// TIA Portal V16 export
// export: Created 2022-11-17T15:49:33.7252465Z, ExportSetting WithDefaults, DisplayName Totally Integrated Automation Portal, DisplayVersion V16 Update 6, DisplayName TIA Portal Version Control Interface, DisplayVersion V16 Update 2, DisplayName TIA Portal Openness, DisplayVersion V16 Update 6, DisplayName SINAMICS Startdrive Advanced, DisplayVersion V16 Update 5, DisplayName SINAMICS Startdrive G130, G150, S120, S150, SINAMICS MV, S210, DisplayVersion V16 Update 5, DisplayName SINAMICS Startdrive G110M, G120, G120C, G120D, G120P, G115D, DisplayVersion V16 Update 5, DisplayName STEP 7 Professional, DisplayVersion V16 Update 6, DisplayName STEP 7 Safety, DisplayVersion V16, DisplayName WinCC Advanced, DisplayVersion V16 Update 6
ORGANIZATION_BLOCK "Main"   // OB1, LAD, ProgramCycle
TITLE = "Main Program Sweep (Cycle)"
{ S7_Optimized_Access := 'TRUE' }
VERSION : 0.1
// stored: AutoNumber false, IsIECCheckEnabled false, SetENOAutomatically false
   VAR_TEMP
      SALDATORE : Bool;
      PORTA : Bool;
      ESAUR_FILM : Bool;
      STR_FASCIA : Bool;
      STR_CORDA : Bool;
      CONTRASTO : Bool;
      PRESSORE : Bool;
      PRESS_RECT : Bool;
      AUTO_CENTR : Bool;
      TOP : Bool;
      BRAKE : Bool;   // Table phase
      PHASE : Bool;   // Table brake
   END_VAR
   VAR_TEMP   // added for the SCL form of the ladder/FBD networks
      _w1 : Bool;
      _w2 : Bool;
      _w3 : Bool;
   END_VAR
BEGIN

REGION Network 1: Bit always on
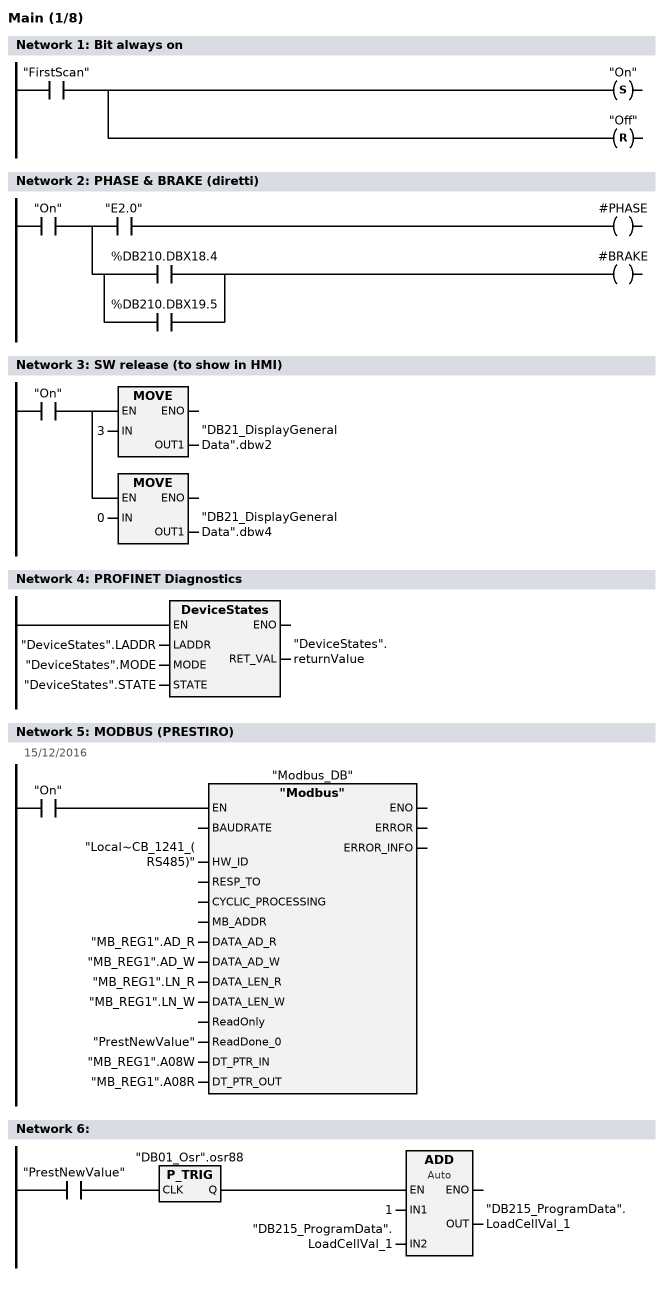
   RUNG wire#powerrail
      Contact( "FirstScan" )
      wire#w1
      S_Coil( "On" )
   END_RUNG
   RUNG wire#w1
      R_Coil( "Off" )
   END_RUNG
   // the same network as SCL:
   IF "FirstScan" THEN
       "On" := TRUE;
       "Off" := FALSE;
   END_IF;
END_REGION

REGION Network 2: PHASE & BRAKE (diretti)
   RUNG wire#powerrail
      Contact( "On" )
      wire#w1
      Contact( "E2.0" )
      Coil( #PHASE )
   END_RUNG
   RUNG wire#w1
      Contact( %DB210.DBX18.4 )
      wire#w2
      Coil( #BRAKE )
   END_RUNG
   RUNG wire#w1
      Contact( %DB210.DBX19.5 )
   END_RUNG wire#w2
   // the same network as SCL:
   #PHASE := "On" AND "E2.0";
   #BRAKE := "On" AND (%DB210.DBX18.4 OR %DB210.DBX19.5);
END_REGION

REGION Network 3: SW release (to show in HMI)
   RUNG wire#powerrail
      Contact( "On" )
      wire#w1
      Move(in := 3, out1 => "DB21_DisplayGeneralData".dbw2)
   END_RUNG
   RUNG wire#w1
      Move(in := 0, out1 => "DB21_DisplayGeneralData".dbw4)
   END_RUNG
   // the same network as SCL:
   IF "On" THEN
       "DB21_DisplayGeneralData".dbw2 := 3;
       "DB21_DisplayGeneralData".dbw4 := 0;
   END_IF;
END_REGION

REGION Network 4: PROFINET Diagnostics
   RUNG wire#powerrail
      DeviceStates(LADDR := "DeviceStates".LADDR, MODE := "DeviceStates".MODE, STATE := "DeviceStates".STATE, Ret_Val => "DeviceStates".returnValue)
   END_RUNG
   // the same network as SCL:
   "DeviceStates".returnValue := DeviceStates(LADDR := "DeviceStates".LADDR,
                           MODE := "DeviceStates".MODE,
                           STATE := "DeviceStates".STATE);
END_REGION

REGION Network 5: MODBUS (PRESTIRO)
   // 15/12/2016
   RUNG wire#powerrail
      Contact( "On" )
      "Modbus_DB"(BAUDRATE :=, HW_ID := "Local~CB_1241_(RS485)", RESP_TO :=, CYCLIC_PROCESSING :=, MB_ADDR :=, DATA_AD_R := "MB_REG1".AD_R, DATA_AD_W := "MB_REG1".AD_W, DATA_LEN_R := "MB_REG1".LN_R, DATA_LEN_W := "MB_REG1".LN_W, ReadOnly :=, ReadDone_0 := "PrestNewValue", DT_PTR_IN := "MB_REG1".A08W, DT_PTR_OUT := "MB_REG1".A08R, ERROR =>, ERROR_INFO =>)
   END_RUNG
   // the same network as SCL:
   IF "On" THEN
       "Modbus_DB"(HW_ID := "Local~CB_1241_(RS485)",   // "Modbus"
                   DATA_AD_R := "MB_REG1".AD_R,
                   DATA_AD_W := "MB_REG1".AD_W,
                   DATA_LEN_R := "MB_REG1".LN_R,
                   DATA_LEN_W := "MB_REG1".LN_W,
                   ReadDone_0 := "PrestNewValue",
                   DT_PTR_IN := "MB_REG1".A08W,
                   DT_PTR_OUT := "MB_REG1".A08R);
   END_IF;
END_REGION

REGION Network 6
   RUNG wire#powerrail
      Contact( "PrestNewValue" )
      P_Trig( "DB01_Osr".osr88 )
      Add(in1 := 1, in2 := "DB215_ProgramData".LoadCellVal_1, out => "DB215_ProgramData".LoadCellVal_1)
   END_RUNG
   // the same network as SCL:
   #_w1 := "PrestNewValue" AND NOT "DB01_Osr".osr88;   // rising edge
   "DB01_Osr".osr88 := "PrestNewValue";
   IF #_w1 THEN "DB215_ProgramData".LoadCellVal_1 := 1 + "DB215_ProgramData".LoadCellVal_1; END_IF;
END_REGION

REGION Network 7: Reset Modbus errors
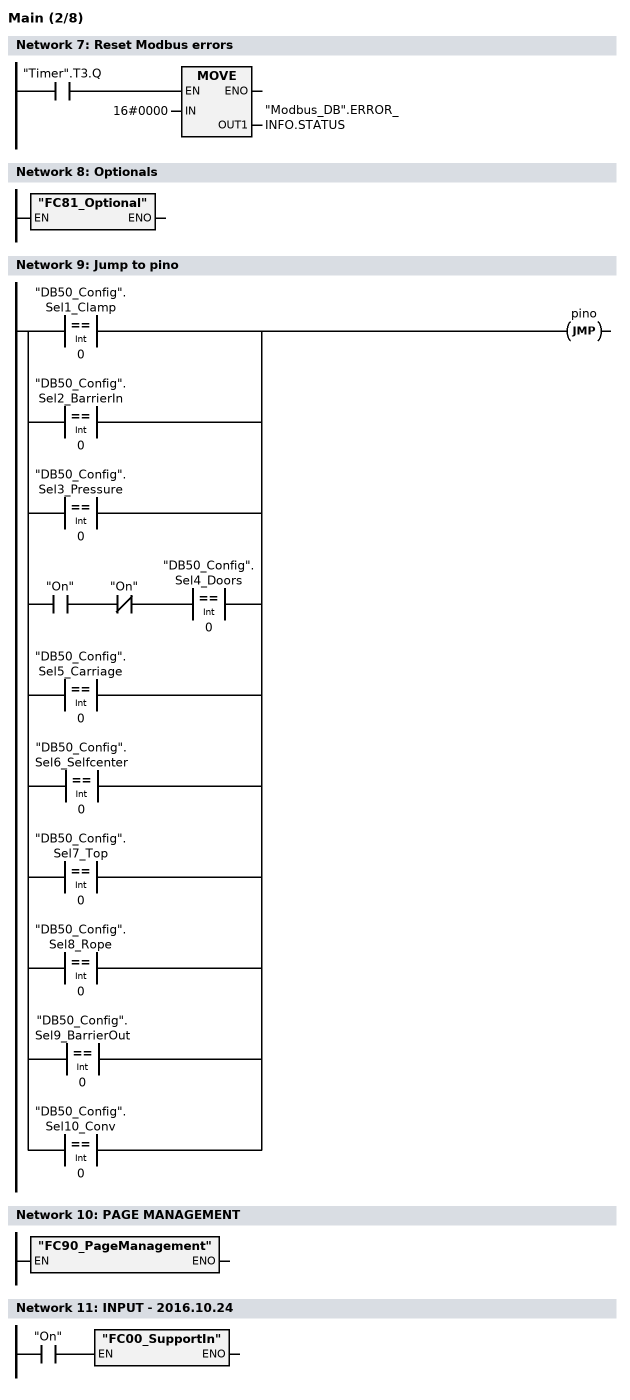
   RUNG wire#powerrail
      Contact( "Timer".T3.Q )
      Move(in := 16#0000, out1 => "Modbus_DB".ERROR_INFO.STATUS)
   END_RUNG
   // the same network as SCL:
   IF "Timer".T3.Q THEN "Modbus_DB".ERROR_INFO.STATUS := 16#0000; END_IF;
END_REGION

REGION Network 8: Optionals
   RUNG wire#powerrail
      "FC81_Optional"()
   END_RUNG
   // the same network as SCL:
   "FC81_Optional"();
END_REGION

REGION Network 9: Jump to pino
   RUNG wire#powerrail
      { S7_Templates := "SrcType := Int" } EQ_Contact(in1 := "DB50_Config".Sel1_Clamp, in2 := 0)
      wire#w1
      JumpCoil( pino )
   END_RUNG
   RUNG wire#powerrail
      { S7_Templates := "SrcType := Int" } EQ_Contact(in1 := "DB50_Config".Sel2_BarrierIn, in2 := 0)
   END_RUNG wire#w1
   RUNG wire#powerrail
      { S7_Templates := "SrcType := Int" } EQ_Contact(in1 := "DB50_Config".Sel3_Pressure, in2 := 0)
   END_RUNG wire#w1
   RUNG wire#powerrail
      Contact( "On" )
      I_Contact( "On" )
      { S7_Templates := "SrcType := Int" } EQ_Contact(in1 := "DB50_Config".Sel4_Doors, in2 := 0)
   END_RUNG wire#w1
   RUNG wire#powerrail
      { S7_Templates := "SrcType := Int" } EQ_Contact(in1 := "DB50_Config".Sel5_Carriage, in2 := 0)
   END_RUNG wire#w1
   RUNG wire#powerrail
      { S7_Templates := "SrcType := Int" } EQ_Contact(in1 := "DB50_Config".Sel6_Selfcenter, in2 := 0)
   END_RUNG wire#w1
   RUNG wire#powerrail
      { S7_Templates := "SrcType := Int" } EQ_Contact(in1 := "DB50_Config".Sel7_Top, in2 := 0)
   END_RUNG wire#w1
   RUNG wire#powerrail
      { S7_Templates := "SrcType := Int" } EQ_Contact(in1 := "DB50_Config".Sel8_Rope, in2 := 0)
   END_RUNG wire#w1
   RUNG wire#powerrail
      { S7_Templates := "SrcType := Int" } EQ_Contact(in1 := "DB50_Config".Sel9_BarrierOut, in2 := 0)
   END_RUNG wire#w1
   RUNG wire#powerrail
      { S7_Templates := "SrcType := Int" } EQ_Contact(in1 := "DB50_Config".Sel10_Conv, in2 := 0)
   END_RUNG wire#w1
   // the same network as SCL:
   IF ("DB50_Config".Sel1_Clamp = 0) OR ("DB50_Config".Sel2_BarrierIn = 0) OR ("DB50_Config".Sel3_Pressure = 0) OR ("On" AND NOT "On" AND ("DB50_Config".Sel4_Doors = 0)) OR ("DB50_Config".Sel5_Carriage = 0) OR ("DB50_Config".Sel6_Selfcenter = 0) OR ("DB50_Config".Sel7_Top = 0) OR ("DB50_Config".Sel8_Rope = 0) OR ("DB50_Config".Sel9_BarrierOut = 0) OR ("DB50_Config".Sel10_Conv = 0) THEN
       GOTO pino;
   END_IF;
END_REGION

REGION Network 10: PAGE MANAGEMENT
   RUNG wire#powerrail
      "FC90_PageManagement"()
   END_RUNG
   // the same network as SCL:
   "FC90_PageManagement"();
END_REGION

REGION Network 11: INPUT - 2016.10.24
   RUNG wire#powerrail
      Contact( "On" )
      "FC00_SupportIn"()
   END_RUNG
   // the same network as SCL:
   IF "On" THEN "FC00_SupportIn"(); END_IF;
END_REGION

REGION Network 12: ACCESSORIES (CONFIGURATION)
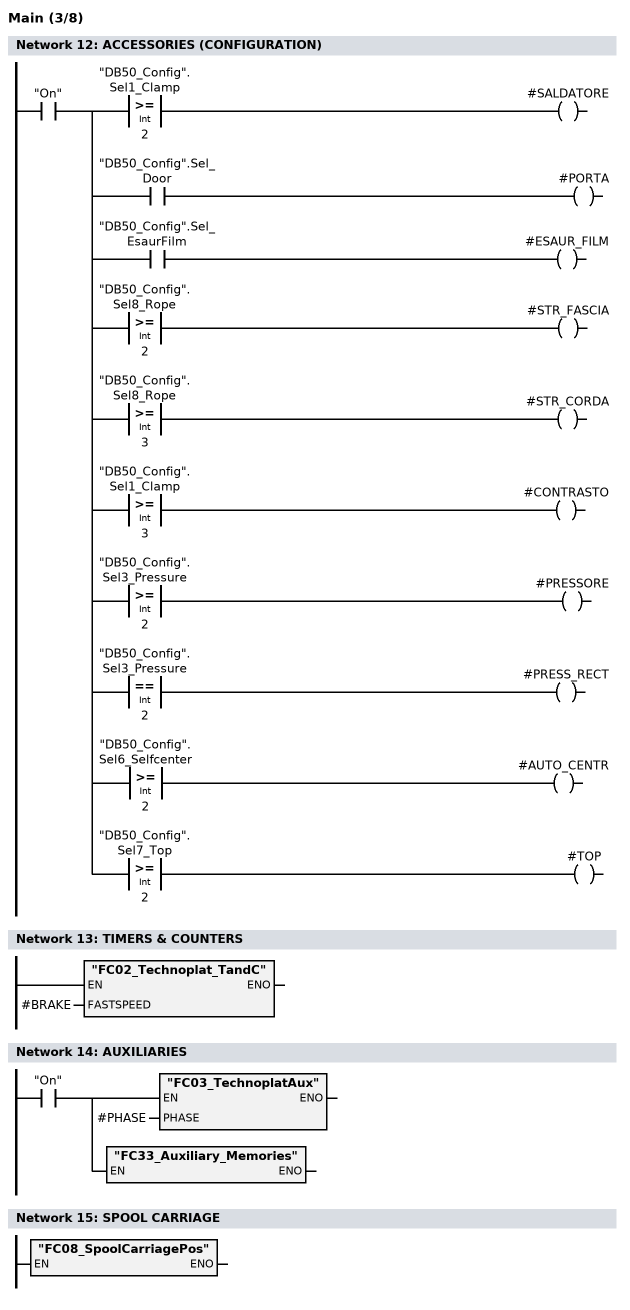
   RUNG wire#powerrail
      Contact( "On" )
      wire#w1
      { S7_Templates := "SrcType := Int" } GE_Contact(in1 := "DB50_Config".Sel1_Clamp, in2 := 2)
      Coil( #SALDATORE )
   END_RUNG
   RUNG wire#w1
      Contact( "DB50_Config".Sel_Door )
      Coil( #PORTA )
   END_RUNG
   RUNG wire#w1
      Contact( "DB50_Config".Sel_EsaurFilm )
      Coil( #ESAUR_FILM )
   END_RUNG
   RUNG wire#w1
      { S7_Templates := "SrcType := Int" } GE_Contact(in1 := "DB50_Config".Sel8_Rope, in2 := 2)
      Coil( #STR_FASCIA )
   END_RUNG
   RUNG wire#w1
      { S7_Templates := "SrcType := Int" } GE_Contact(in1 := "DB50_Config".Sel8_Rope, in2 := 3)
      Coil( #STR_CORDA )
   END_RUNG
   RUNG wire#w1
      { S7_Templates := "SrcType := Int" } GE_Contact(in1 := "DB50_Config".Sel1_Clamp, in2 := 3)
      Coil( #CONTRASTO )
   END_RUNG
   RUNG wire#w1
      { S7_Templates := "SrcType := Int" } GE_Contact(in1 := "DB50_Config".Sel3_Pressure, in2 := 2)
      Coil( #PRESSORE )
   END_RUNG
   RUNG wire#w1
      { S7_Templates := "SrcType := Int" } EQ_Contact(in1 := "DB50_Config".Sel3_Pressure, in2 := 2)
      Coil( #PRESS_RECT )
   END_RUNG
   RUNG wire#w1
      { S7_Templates := "SrcType := Int" } GE_Contact(in1 := "DB50_Config".Sel6_Selfcenter, in2 := 2)
      Coil( #AUTO_CENTR )
   END_RUNG
   RUNG wire#w1
      { S7_Templates := "SrcType := Int" } GE_Contact(in1 := "DB50_Config".Sel7_Top, in2 := 2)
      Coil( #TOP )
   END_RUNG
   // the same network as SCL:
   #SALDATORE := "On" AND ("DB50_Config".Sel1_Clamp >= 2);
   #PORTA := "On" AND "DB50_Config".Sel_Door;
   #ESAUR_FILM := "On" AND "DB50_Config".Sel_EsaurFilm;
   #STR_FASCIA := "On" AND ("DB50_Config".Sel8_Rope >= 2);
   #STR_CORDA := "On" AND ("DB50_Config".Sel8_Rope >= 3);
   #CONTRASTO := "On" AND ("DB50_Config".Sel1_Clamp >= 3);
   #PRESSORE := "On" AND ("DB50_Config".Sel3_Pressure >= 2);
   #PRESS_RECT := "On" AND ("DB50_Config".Sel3_Pressure = 2);
   #AUTO_CENTR := "On" AND ("DB50_Config".Sel6_Selfcenter >= 2);
   #TOP := "On" AND ("DB50_Config".Sel7_Top >= 2);
END_REGION

REGION Network 13: TIMERS & COUNTERS
   RUNG wire#powerrail
      "FC02_Technoplat_TandC"(FASTSPEED := #BRAKE)
   END_RUNG
   // the same network as SCL:
   "FC02_Technoplat_TandC"(FASTSPEED := #BRAKE);
END_REGION

REGION Network 14: AUXILIARIES
   RUNG wire#powerrail
      Contact( "On" )
      wire#w1
      "FC03_TechnoplatAux"(PHASE := #PHASE)
   END_RUNG
   RUNG wire#w1
      "FC33_Auxiliary_Memories"()
   END_RUNG
   // the same network as SCL:
   #_w1 := "On";
   IF #_w1 THEN
       "FC03_TechnoplatAux"(PHASE := #PHASE);
       "FC33_Auxiliary_Memories"();
   END_IF;
END_REGION

REGION Network 15: SPOOL CARRIAGE
   RUNG wire#powerrail
      "FC08_SpoolCarriagePos"()
   END_RUNG
   // the same network as SCL:
   "FC08_SpoolCarriagePos"();
END_REGION

REGION Network 16: ROTATION TABLE
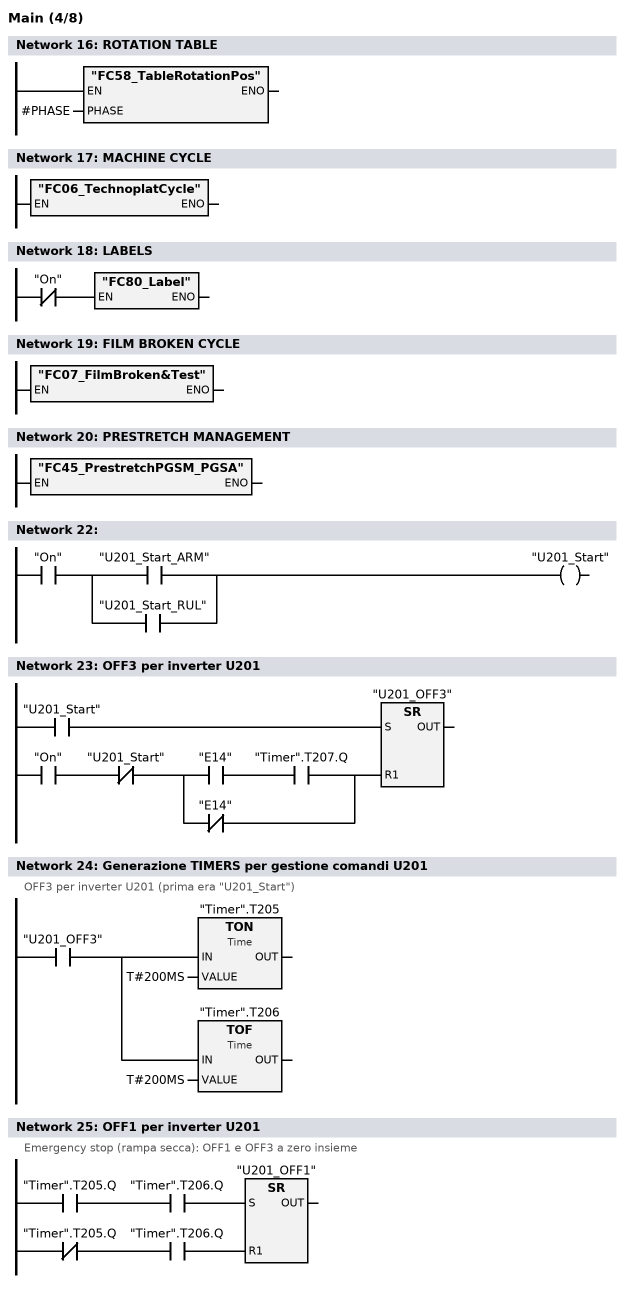
   RUNG wire#powerrail
      "FC58_TableRotationPos"(PHASE := #PHASE)
   END_RUNG
   // the same network as SCL:
   "FC58_TableRotationPos"(PHASE := #PHASE);
END_REGION

REGION Network 17: MACHINE CYCLE
   RUNG wire#powerrail
      "FC06_TechnoplatCycle"()
   END_RUNG
   // the same network as SCL:
   "FC06_TechnoplatCycle"();
END_REGION

REGION Network 18: LABELS
   RUNG wire#powerrail
      I_Contact( "On" )
      "FC80_Label"()
   END_RUNG
   // the same network as SCL:
   IF NOT "On" THEN "FC80_Label"(); END_IF;
END_REGION

REGION Network 19: FILM BROKEN CYCLE
   RUNG wire#powerrail
      "FC07_FilmBroken&Test"()
   END_RUNG
   // the same network as SCL:
   "FC07_FilmBroken&Test"();
END_REGION

REGION Network 20: PRESTRETCH MANAGEMENT
   RUNG wire#powerrail
      "FC45_PrestretchPGSM_PGSA"()
   END_RUNG
   // the same network as SCL:
   "FC45_PrestretchPGSM_PGSA"();
END_REGION

REGION Network 21: - - - GESTIONE INVERTER PROFINET - - -
END_REGION

REGION Network 22
   RUNG wire#powerrail
      Contact( "On" )
      wire#w1
      Contact( "U201_Start_ARM" )
      wire#w2
      Coil( "U201_Start" )
   END_RUNG
   RUNG wire#w1
      Contact( "U201_Start_RUL" )
   END_RUNG wire#w2
   // the same network as SCL:
   "U201_Start" := "On" AND ("U201_Start_ARM" OR "U201_Start_RUL");
END_REGION

REGION Network 23: OFF3 per inverter U201
   RUNG wire#powerrail
      Contact( "U201_Start" )
      S_SR(operand := "U201_OFF3", r1 := wire#w2)
   END_RUNG
   RUNG wire#powerrail
      Contact( "On" )
      I_Contact( "U201_Start" )
      wire#w1
      Contact( "E14" )
      Contact( "Timer".T207.Q )
   END_RUNG wire#w2
   RUNG wire#w1
      I_Contact( "E14" )
   END_RUNG wire#w2
   // the same network as SCL:
   IF "U201_Start" THEN
       "U201_OFF3" := TRUE;   // SR flip-flop
   END_IF;
   IF "On" AND NOT "U201_Start" AND (("E14" AND "Timer".T207.Q) OR NOT "E14") THEN
       "U201_OFF3" := FALSE;
   END_IF;
END_REGION

REGION Network 24: Generazione TIMERS per gestione comandi U201
   // OFF3 per inverter U201 (prima era "U201_Start")
   "Timer".T205.TON(IN := "U201_OFF3", PT := T#200MS);   // TON coil
   "Timer".T206.TOF(IN := "U201_OFF3", PT := T#200MS);   // TOF coil
END_REGION

REGION Network 25: OFF1 per inverter U201
   // Emergency stop (rampa secca): OFF1 e OFF3 a zero insieme
   RUNG wire#powerrail
      Contact( "Timer".T205.Q )
      Contact( "Timer".T206.Q )
      S_SR(operand := "U201_OFF1", r1 := wire#w1)
   END_RUNG
   RUNG wire#powerrail
      I_Contact( "Timer".T205.Q )
      Contact( "Timer".T206.Q )
   END_RUNG wire#w1
   // the same network as SCL:
   IF "Timer".T205.Q AND "Timer".T206.Q THEN
       "U201_OFF1" := TRUE;   // SR flip-flop
   END_IF;
   IF NOT "Timer".T205.Q AND "Timer".T206.Q THEN "U201_OFF1" := FALSE; END_IF;
END_REGION

REGION Network 26: U201 - ROTAZIONE + CM
   // "U201_OFF1"/"U201_OFF3"
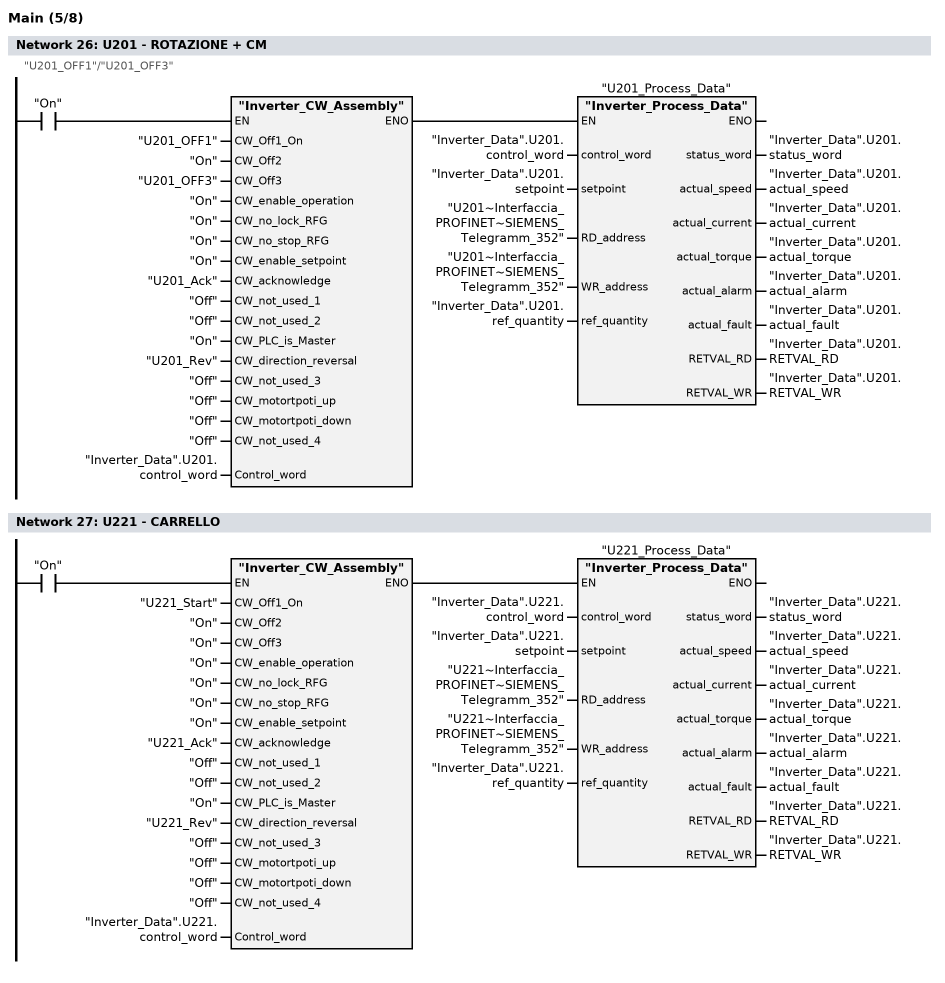
   RUNG wire#powerrail
      Contact( "On" )
      "Inverter_CW_Assembly"(CW_Off1_On := "U201_OFF1", CW_Off2 := "On", CW_Off3 := "U201_OFF3", CW_enable_operation := "On", CW_no_lock_RFG := "On", CW_no_stop_RFG := "On", CW_enable_setpoint := "On", CW_acknowledge := "U201_Ack", CW_not_used_1 := "Off", CW_not_used_2 := "Off", CW_PLC_is_Master := "On", CW_direction_reversal := "U201_Rev", CW_not_used_3 := "Off", CW_motortpoti_up := "Off", CW_motortpoti_down := "Off", CW_not_used_4 := "Off", Control_word := "Inverter_Data".U201.control_word)
      "U201_Process_Data"(control_word := "Inverter_Data".U201.control_word, setpoint := "Inverter_Data".U201.setpoint, RD_address := "U201~Interfaccia_PROFINET~SIEMENS_Telegramm_352", WR_address := "U201~Interfaccia_PROFINET~SIEMENS_Telegramm_352", ref_quantity := "Inverter_Data".U201.ref_quantity, status_word => "Inverter_Data".U201.status_word, actual_speed => "Inverter_Data".U201.actual_speed, actual_current => "Inverter_Data".U201.actual_current, actual_torque => "Inverter_Data".U201.actual_torque, actual_alarm => "Inverter_Data".U201.actual_alarm, actual_fault => "Inverter_Data".U201.actual_fault, RETVAL_RD => "Inverter_Data".U201.RETVAL_RD, RETVAL_WR => "Inverter_Data".U201.RETVAL_WR)
   END_RUNG
   // the same network as SCL:
   "Inverter_CW_Assembly"(EN := "On",
                          CW_Off1_On := "U201_OFF1",
                          CW_Off2 := "On",
                          CW_Off3 := "U201_OFF3",
                          CW_enable_operation := "On",
                          CW_no_lock_RFG := "On",
                          CW_no_stop_RFG := "On",
                          CW_enable_setpoint := "On",
                          CW_acknowledge := "U201_Ack",
                          CW_not_used_1 := "Off",
                          CW_not_used_2 := "Off",
                          CW_PLC_is_Master := "On",
                          CW_direction_reversal := "U201_Rev",
                          CW_not_used_3 := "Off",
                          CW_motortpoti_up := "Off",
                          CW_motortpoti_down := "Off",
                          CW_not_used_4 := "Off",
                          Control_word := "Inverter_Data".U201.control_word,
                          ENO => #_w1);
   IF #_w1 THEN
       "U201_Process_Data"(control_word := "Inverter_Data".U201.control_word,   // "Inverter_Process_Data"
                           setpoint := "Inverter_Data".U201.setpoint,
                           RD_address := "U201~Interfaccia_PROFINET~SIEMENS_Telegramm_352",
                           WR_address := "U201~Interfaccia_PROFINET~SIEMENS_Telegramm_352",
                           ref_quantity := "Inverter_Data".U201.ref_quantity,
                           status_word => "Inverter_Data".U201.status_word,
                           actual_speed => "Inverter_Data".U201.actual_speed,
                           actual_current => "Inverter_Data".U201.actual_current,
                           actual_torque => "Inverter_Data".U201.actual_torque,
                           actual_alarm => "Inverter_Data".U201.actual_alarm,
                           actual_fault => "Inverter_Data".U201.actual_fault,
                           RETVAL_RD => "Inverter_Data".U201.RETVAL_RD,
                           RETVAL_WR => "Inverter_Data".U201.RETVAL_WR);
   END_IF;
END_REGION

REGION Network 27: U221 - CARRELLO
   RUNG wire#powerrail
      Contact( "On" )
      "Inverter_CW_Assembly"(CW_Off1_On := "U221_Start", CW_Off2 := "On", CW_Off3 := "On", CW_enable_operation := "On", CW_no_lock_RFG := "On", CW_no_stop_RFG := "On", CW_enable_setpoint := "On", CW_acknowledge := "U221_Ack", CW_not_used_1 := "Off", CW_not_used_2 := "Off", CW_PLC_is_Master := "On", CW_direction_reversal := "U221_Rev", CW_not_used_3 := "Off", CW_motortpoti_up := "Off", CW_motortpoti_down := "Off", CW_not_used_4 := "Off", Control_word := "Inverter_Data".U221.control_word)
      "U221_Process_Data"(control_word := "Inverter_Data".U221.control_word, setpoint := "Inverter_Data".U221.setpoint, RD_address := "U221~Interfaccia_PROFINET~SIEMENS_Telegramm_352", WR_address := "U221~Interfaccia_PROFINET~SIEMENS_Telegramm_352", ref_quantity := "Inverter_Data".U221.ref_quantity, status_word => "Inverter_Data".U221.status_word, actual_speed => "Inverter_Data".U221.actual_speed, actual_current => "Inverter_Data".U221.actual_current, actual_torque => "Inverter_Data".U221.actual_torque, actual_alarm => "Inverter_Data".U221.actual_alarm, actual_fault => "Inverter_Data".U221.actual_fault, RETVAL_RD => "Inverter_Data".U221.RETVAL_RD, RETVAL_WR => "Inverter_Data".U221.RETVAL_WR)
   END_RUNG
   // the same network as SCL:
   "Inverter_CW_Assembly"(EN := "On",
                          CW_Off1_On := "U221_Start",
                          CW_Off2 := "On",
                          CW_Off3 := "On",
                          CW_enable_operation := "On",
                          CW_no_lock_RFG := "On",
                          CW_no_stop_RFG := "On",
                          CW_enable_setpoint := "On",
                          CW_acknowledge := "U221_Ack",
                          CW_not_used_1 := "Off",
                          CW_not_used_2 := "Off",
                          CW_PLC_is_Master := "On",
                          CW_direction_reversal := "U221_Rev",
                          CW_not_used_3 := "Off",
                          CW_motortpoti_up := "Off",
                          CW_motortpoti_down := "Off",
                          CW_not_used_4 := "Off",
                          Control_word := "Inverter_Data".U221.control_word,
                          ENO => #_w1);
   IF #_w1 THEN
       "U221_Process_Data"(control_word := "Inverter_Data".U221.control_word,   // "Inverter_Process_Data"
                           setpoint := "Inverter_Data".U221.setpoint,
                           RD_address := "U221~Interfaccia_PROFINET~SIEMENS_Telegramm_352",
                           WR_address := "U221~Interfaccia_PROFINET~SIEMENS_Telegramm_352",
                           ref_quantity := "Inverter_Data".U221.ref_quantity,
                           status_word => "Inverter_Data".U221.status_word,
                           actual_speed => "Inverter_Data".U221.actual_speed,
                           actual_current => "Inverter_Data".U221.actual_current,
                           actual_torque => "Inverter_Data".U221.actual_torque,
                           actual_alarm => "Inverter_Data".U221.actual_alarm,
                           actual_fault => "Inverter_Data".U221.actual_fault,
                           RETVAL_RD => "Inverter_Data".U221.RETVAL_RD,
                           RETVAL_WR => "Inverter_Data".U221.RETVAL_WR);
   END_IF;
END_REGION

REGION Network 28: U241 - PRESTIRO (VELOCE)
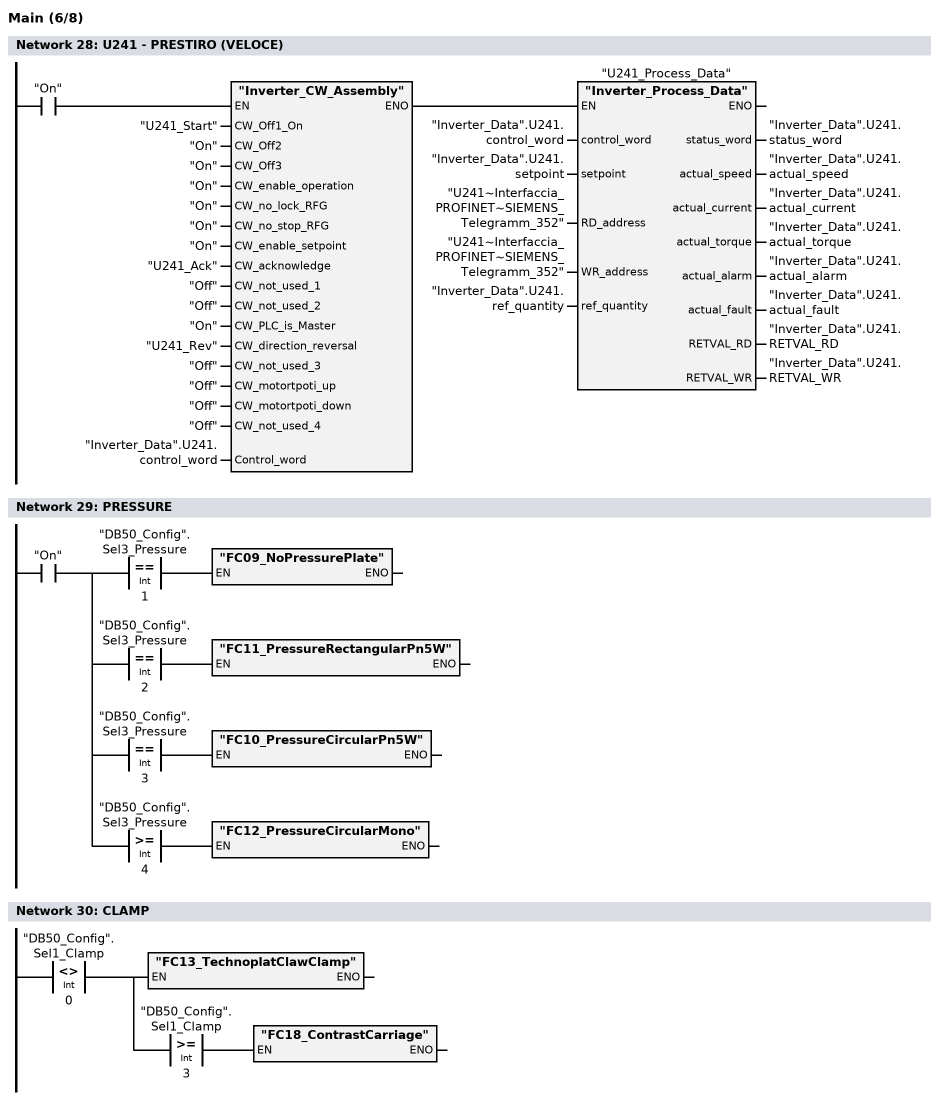
   RUNG wire#powerrail
      Contact( "On" )
      "Inverter_CW_Assembly"(CW_Off1_On := "U241_Start", CW_Off2 := "On", CW_Off3 := "On", CW_enable_operation := "On", CW_no_lock_RFG := "On", CW_no_stop_RFG := "On", CW_enable_setpoint := "On", CW_acknowledge := "U241_Ack", CW_not_used_1 := "Off", CW_not_used_2 := "Off", CW_PLC_is_Master := "On", CW_direction_reversal := "U241_Rev", CW_not_used_3 := "Off", CW_motortpoti_up := "Off", CW_motortpoti_down := "Off", CW_not_used_4 := "Off", Control_word := "Inverter_Data".U241.control_word)
      "U241_Process_Data"(control_word := "Inverter_Data".U241.control_word, setpoint := "Inverter_Data".U241.setpoint, RD_address := "U241~Interfaccia_PROFINET~SIEMENS_Telegramm_352", WR_address := "U241~Interfaccia_PROFINET~SIEMENS_Telegramm_352", ref_quantity := "Inverter_Data".U241.ref_quantity, status_word => "Inverter_Data".U241.status_word, actual_speed => "Inverter_Data".U241.actual_speed, actual_current => "Inverter_Data".U241.actual_current, actual_torque => "Inverter_Data".U241.actual_torque, actual_alarm => "Inverter_Data".U241.actual_alarm, actual_fault => "Inverter_Data".U241.actual_fault, RETVAL_RD => "Inverter_Data".U241.RETVAL_RD, RETVAL_WR => "Inverter_Data".U241.RETVAL_WR)
   END_RUNG
   // the same network as SCL:
   "Inverter_CW_Assembly"(EN := "On",
                          CW_Off1_On := "U241_Start",
                          CW_Off2 := "On",
                          CW_Off3 := "On",
                          CW_enable_operation := "On",
                          CW_no_lock_RFG := "On",
                          CW_no_stop_RFG := "On",
                          CW_enable_setpoint := "On",
                          CW_acknowledge := "U241_Ack",
                          CW_not_used_1 := "Off",
                          CW_not_used_2 := "Off",
                          CW_PLC_is_Master := "On",
                          CW_direction_reversal := "U241_Rev",
                          CW_not_used_3 := "Off",
                          CW_motortpoti_up := "Off",
                          CW_motortpoti_down := "Off",
                          CW_not_used_4 := "Off",
                          Control_word := "Inverter_Data".U241.control_word,
                          ENO => #_w1);
   IF #_w1 THEN
       "U241_Process_Data"(control_word := "Inverter_Data".U241.control_word,   // "Inverter_Process_Data"
                           setpoint := "Inverter_Data".U241.setpoint,
                           RD_address := "U241~Interfaccia_PROFINET~SIEMENS_Telegramm_352",
                           WR_address := "U241~Interfaccia_PROFINET~SIEMENS_Telegramm_352",
                           ref_quantity := "Inverter_Data".U241.ref_quantity,
                           status_word => "Inverter_Data".U241.status_word,
                           actual_speed => "Inverter_Data".U241.actual_speed,
                           actual_current => "Inverter_Data".U241.actual_current,
                           actual_torque => "Inverter_Data".U241.actual_torque,
                           actual_alarm => "Inverter_Data".U241.actual_alarm,
                           actual_fault => "Inverter_Data".U241.actual_fault,
                           RETVAL_RD => "Inverter_Data".U241.RETVAL_RD,
                           RETVAL_WR => "Inverter_Data".U241.RETVAL_WR);
   END_IF;
END_REGION

REGION Network 29: PRESSURE
   RUNG wire#powerrail
      Contact( "On" )
      wire#w1
      { S7_Templates := "SrcType := Int" } EQ_Contact(in1 := "DB50_Config".Sel3_Pressure, in2 := 1)
      "FC09_NoPressurePlate"()
   END_RUNG
   RUNG wire#w1
      { S7_Templates := "SrcType := Int" } EQ_Contact(in1 := "DB50_Config".Sel3_Pressure, in2 := 2)
      "FC11_PressureRectangularPn5W"()
   END_RUNG
   RUNG wire#w1
      { S7_Templates := "SrcType := Int" } EQ_Contact(in1 := "DB50_Config".Sel3_Pressure, in2 := 3)
      "FC10_PressureCircularPn5W"()
   END_RUNG
   RUNG wire#w1
      { S7_Templates := "SrcType := Int" } GE_Contact(in1 := "DB50_Config".Sel3_Pressure, in2 := 4)
      "FC12_PressureCircularMono"()
   END_RUNG
   // the same network as SCL:
   #_w1 := "On";
   IF "On" AND ("DB50_Config".Sel3_Pressure = 1) THEN "FC09_NoPressurePlate"(); END_IF;
   IF #_w1 AND ("DB50_Config".Sel3_Pressure = 2) THEN "FC11_PressureRectangularPn5W"(); END_IF;
   IF #_w1 AND ("DB50_Config".Sel3_Pressure = 3) THEN "FC10_PressureCircularPn5W"(); END_IF;
   IF #_w1 AND ("DB50_Config".Sel3_Pressure >= 4) THEN "FC12_PressureCircularMono"(); END_IF;
END_REGION

REGION Network 30: CLAMP
   RUNG wire#powerrail
      { S7_Templates := "SrcType := Int" } NE_Contact(in1 := "DB50_Config".Sel1_Clamp, in2 := 0)
      wire#w1
      "FC13_TechnoplatClawClamp"()
   END_RUNG
   RUNG wire#w1
      { S7_Templates := "SrcType := Int" } GE_Contact(in1 := "DB50_Config".Sel1_Clamp, in2 := 3)
      "FC18_ContrastCarriage"()
   END_RUNG
   // the same network as SCL:
   #_w1 := "DB50_Config".Sel1_Clamp <> 0;
   IF #_w1 THEN "FC13_TechnoplatClawClamp"(); END_IF;
   IF #_w1 AND ("DB50_Config".Sel1_Clamp >= 3) THEN "FC18_ContrastCarriage"(); END_IF;
END_REGION

REGION Network 31: Lifter selection
END_REGION

REGION Network 32: TOP
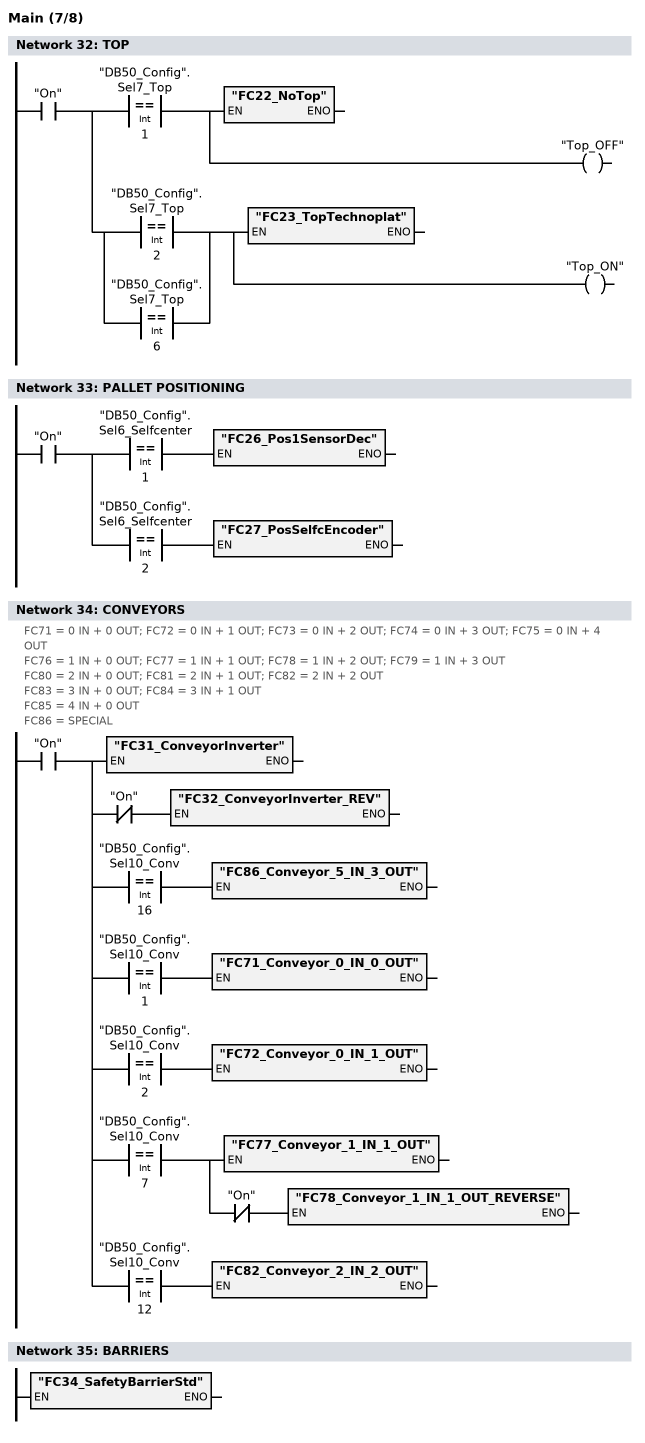
   RUNG wire#powerrail
      Contact( "On" )
      wire#w1
      { S7_Templates := "SrcType := Int" } EQ_Contact(in1 := "DB50_Config".Sel7_Top, in2 := 1)
      wire#w2
      "FC22_NoTop"()
   END_RUNG
   RUNG wire#w2
      Coil( "Top_OFF" )
   END_RUNG
   RUNG wire#w1
      { S7_Templates := "SrcType := Int" } EQ_Contact(in1 := "DB50_Config".Sel7_Top, in2 := 2)
      wire#w3
      "FC23_TopTechnoplat"()
   END_RUNG
   RUNG wire#w1
      { S7_Templates := "SrcType := Int" } EQ_Contact(in1 := "DB50_Config".Sel7_Top, in2 := 6)
   END_RUNG wire#w3
   RUNG wire#w3
      Coil( "Top_ON" )
   END_RUNG
   // the same network as SCL:
   #_w1 := "On" AND ("DB50_Config".Sel7_Top = 1);
   #_w2 := "On";
   IF #_w1 THEN "FC22_NoTop"(); END_IF;
   "Top_OFF" := #_w1;
   #_w3 := #_w2 AND (("DB50_Config".Sel7_Top = 2) OR ("DB50_Config".Sel7_Top = 6));
   IF #_w3 THEN "FC23_TopTechnoplat"(); END_IF;
   "Top_ON" := #_w3;
END_REGION

REGION Network 33: PALLET POSITIONING
   RUNG wire#powerrail
      Contact( "On" )
      wire#w1
      { S7_Templates := "SrcType := Int" } EQ_Contact(in1 := "DB50_Config".Sel6_Selfcenter, in2 := 1)
      "FC26_Pos1SensorDec"()
   END_RUNG
   RUNG wire#w1
      { S7_Templates := "SrcType := Int" } EQ_Contact(in1 := "DB50_Config".Sel6_Selfcenter, in2 := 2)
      "FC27_PosSelfcEncoder"()
   END_RUNG
   // the same network as SCL:
   #_w1 := "On";
   IF "On" AND ("DB50_Config".Sel6_Selfcenter = 1) THEN "FC26_Pos1SensorDec"(); END_IF;
   IF #_w1 AND ("DB50_Config".Sel6_Selfcenter = 2) THEN "FC27_PosSelfcEncoder"(); END_IF;
END_REGION

REGION Network 34: CONVEYORS
   // FC71 = 0 IN + 0 OUT; FC72 = 0 IN + 1 OUT; FC73 = 0 IN + 2 OUT; FC74 = 0 IN + 3 OUT; FC75 = 0 IN + 4 OUT
   // FC76 = 1 IN + 0 OUT; FC77 = 1 IN + 1 OUT; FC78 = 1 IN + 2 OUT; FC79 = 1 IN + 3 OUT
   // FC80 = 2 IN + 0 OUT; FC81 = 2 IN + 1 OUT; FC82 = 2 IN + 2 OUT
   // FC83 = 3 IN + 0 OUT; FC84 = 3 IN + 1 OUT
   // FC85 = 4 IN + 0 OUT
   // FC86 = SPECIAL
   RUNG wire#powerrail
      Contact( "On" )
      wire#w1
      "FC31_ConveyorInverter"()
   END_RUNG
   RUNG wire#w1
      I_Contact( "On" )
      "FC32_ConveyorInverter_REV"()
   END_RUNG
   RUNG wire#w1
      { S7_Templates := "SrcType := Int" } EQ_Contact(in1 := "DB50_Config".Sel10_Conv, in2 := 16)
      "FC86_Conveyor_5_IN_3_OUT"()
   END_RUNG
   RUNG wire#w1
      { S7_Templates := "SrcType := Int" } EQ_Contact(in1 := "DB50_Config".Sel10_Conv, in2 := 1)
      "FC71_Conveyor_0_IN_0_OUT"()
   END_RUNG
   RUNG wire#w1
      { S7_Templates := "SrcType := Int" } EQ_Contact(in1 := "DB50_Config".Sel10_Conv, in2 := 2)
      "FC72_Conveyor_0_IN_1_OUT"()
   END_RUNG
   RUNG wire#w1
      { S7_Templates := "SrcType := Int" } EQ_Contact(in1 := "DB50_Config".Sel10_Conv, in2 := 7)
      wire#w2
      "FC77_Conveyor_1_IN_1_OUT"()
   END_RUNG
   RUNG wire#w2
      I_Contact( "On" )
      "FC78_Conveyor_1_IN_1_OUT_REVERSE"()
   END_RUNG
   RUNG wire#w1
      { S7_Templates := "SrcType := Int" } EQ_Contact(in1 := "DB50_Config".Sel10_Conv, in2 := 12)
      "FC82_Conveyor_2_IN_2_OUT"()
   END_RUNG
   // the same network as SCL:
   #_w1 := "On";
   IF #_w1 THEN "FC31_ConveyorInverter"(); END_IF;
   IF #_w1 AND NOT "On" THEN "FC32_ConveyorInverter_REV"(); END_IF;
   IF #_w1 AND ("DB50_Config".Sel10_Conv = 16) THEN "FC86_Conveyor_5_IN_3_OUT"(); END_IF;
   IF #_w1 AND ("DB50_Config".Sel10_Conv = 1) THEN "FC71_Conveyor_0_IN_0_OUT"(); END_IF;
   IF #_w1 AND ("DB50_Config".Sel10_Conv = 2) THEN "FC72_Conveyor_0_IN_1_OUT"(); END_IF;
   #_w2 := #_w1 AND ("DB50_Config".Sel10_Conv = 7);
   IF #_w2 THEN "FC77_Conveyor_1_IN_1_OUT"(); END_IF;
   IF #_w2 AND NOT "On" THEN "FC78_Conveyor_1_IN_1_OUT_REVERSE"(); END_IF;
   IF #_w1 AND ("DB50_Config".Sel10_Conv = 12) THEN "FC82_Conveyor_2_IN_2_OUT"(); END_IF;
END_REGION

REGION Network 35: BARRIERS
   RUNG wire#powerrail
      "FC34_SafetyBarrierStd"()
   END_RUNG
   // the same network as SCL:
   "FC34_SafetyBarrierStd"();
END_REGION

REGION Network 36: MULTIPROGRAM
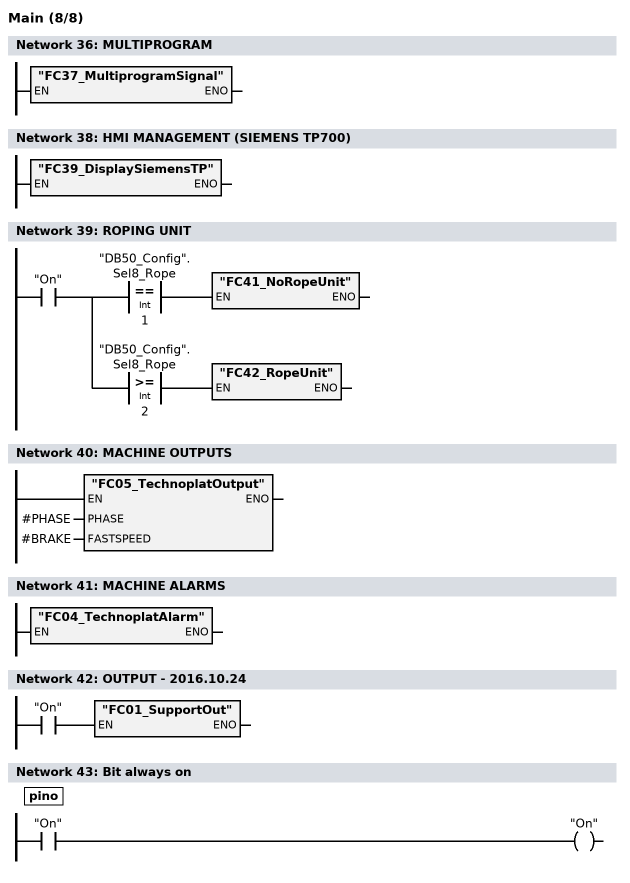
   RUNG wire#powerrail
      "FC37_MultiprogramSignal"()
   END_RUNG
   // the same network as SCL:
   "FC37_MultiprogramSignal"();
END_REGION

REGION Network 37: Incomplete pallet
END_REGION

REGION Network 38: HMI MANAGEMENT (SIEMENS TP700)
   RUNG wire#powerrail
      "FC39_DisplaySiemensTP"()
   END_RUNG
   // the same network as SCL:
   "FC39_DisplaySiemensTP"();
END_REGION

REGION Network 39: ROPING UNIT
   RUNG wire#powerrail
      Contact( "On" )
      wire#w1
      { S7_Templates := "SrcType := Int" } EQ_Contact(in1 := "DB50_Config".Sel8_Rope, in2 := 1)
      "FC41_NoRopeUnit"()
   END_RUNG
   RUNG wire#w1
      { S7_Templates := "SrcType := Int" } GE_Contact(in1 := "DB50_Config".Sel8_Rope, in2 := 2)
      "FC42_RopeUnit"()
   END_RUNG
   // the same network as SCL:
   #_w1 := "On";
   IF "On" AND ("DB50_Config".Sel8_Rope = 1) THEN "FC41_NoRopeUnit"(); END_IF;
   IF #_w1 AND ("DB50_Config".Sel8_Rope >= 2) THEN "FC42_RopeUnit"(); END_IF;
END_REGION

REGION Network 40: MACHINE OUTPUTS
   RUNG wire#powerrail
      "FC05_TechnoplatOutput"(PHASE := #PHASE, FASTSPEED := #BRAKE)
   END_RUNG
   // the same network as SCL:
   "FC05_TechnoplatOutput"(PHASE := #PHASE, FASTSPEED := #BRAKE);
END_REGION

REGION Network 41: MACHINE ALARMS
   RUNG wire#powerrail
      "FC04_TechnoplatAlarm"()
   END_RUNG
   // the same network as SCL:
   "FC04_TechnoplatAlarm"();
END_REGION

REGION Network 42: OUTPUT - 2016.10.24
   RUNG wire#powerrail
      Contact( "On" )
      "FC01_SupportOut"()
   END_RUNG
   // the same network as SCL:
   IF "On" THEN "FC01_SupportOut"(); END_IF;
END_REGION

REGION Network 43: Bit always on
   Label( pino )
   RUNG wire#powerrail
      Contact( "On" )
      Coil( "On" )
   END_RUNG
   // the same network as SCL:
   pino:
   "On" := "On";
END_REGION
END_ORGANIZATION_BLOCK
